{attribute 'qualified_only'}
VAR_GLOBAL
    {attribute 'pytmc' := 'pv: PLC:RIX:MOTION:ARB:01'}
    fbArbiter1: FB_Arbiter(1);
    {attribute 'pytmc' := 'pv: PLC:RIX:MOTION:ARB:02'}
    fbArbiter2: FB_Arbiter(2);

    // For devices between the mirror and the stopper
    {attribute 'pytmc' := 'pv: PLC:RIX:MOTION:FFO:01'}
    {attribute 'TcLinkTo' := '.q_xFastFaultOut:=TIIB[PMPS_FFO]^Channel 1^Output'}
    fbFastFaultOutput1: FB_HardwareFFOutput := (bAutoReset := TRUE, i_sNetID:='172.21.42.126.1.1');

    // For devices after the stopper
    {attribute 'pytmc' := 'pv: PLC:RIX:MOTION:FFO:02'}
    {attribute 'TcLinkTo' := '.q_xFastFaultOut:=TIIB[PMPS_FFO]^Channel 2^Output'}
    fbFastFaultOutput2: FB_HardwareFFOutput := (bAutoReset := TRUE, i_sNetID:='172.21.42.126.1.1');

    fbAtomicMass : FB_AtomicMass;
    fbAttenuatorElementDensity : FB_AttenuatorElementDensity;

    (* Photon energy comes from the arbiter (see PMPS_PRE.IO Inputs.rPhotonEnergy!) *)
	{attribute 'pytmc' := 'pv: PLC:RIX:MOTION:PhotonEnergy'}
    fPhotonEnergy_eV AT %I* : REAL;
	{attribute 'pytmc' := 'pv: PLC:RIX:MOTION:PMPS:ReqTrans'}
	rReqTrans AT %I*		: ARRAY [1..PMPS_GVL.AUX_ATTENUATORS] OF ST_PMPS_Attenuator_IO;
	{attribute 'pytmc' := 'pv: PLC:RIX:MOTION:PMPS:CurTrans'}
	rCurTrans AT %Q*		: ARRAY [1..PMPS_GVL.AUX_ATTENUATORS] OF ST_PMPS_Attenuator_IO;
	
END_VAR

VAR_GLOBAL CONSTANT
    iFiltersPerSATTBlade : INT := 8;
END_VAR

(* stored: Version 1.1.0.1, ProductVersion 3.1.4022.18
   GVL GVL: Id {4e3a33fd-2c1d-4689-9132-04dc3cd973dd} *)
